// TwinCAT 3 PLC project Untitled1
// ProgramVersion: 3.1.4022.4
// libraries:
//   Tc2_MC2, * (Beckhoff Automation GmbH)
//   Tc2_Standard, * (Beckhoff Automation GmbH)
//   Tc2_System, * (Beckhoff Automation GmbH)
//   Tc3_Module, * (Beckhoff Automation GmbH)
// project tree:
//   GVLs/ GVL_IO.TcGVL
//   / PlcTask.TcTTO
//   POUs/ FB_Control.TcPOU, FB_Motion.TcPOU, MAIN.TcPOU
// real-time tasks:
//   TASK PlcTask: cycle T#10ms, priority 20, ADS port 350
// motion (NC):
//   TASK NC-Task 1 SAF: cycle T#2ms, priority 4, ADS port 501
//   TASK NC-Task 1 SVB: cycle T#10ms, priority 8, ADS port 511
//   AXIS Axis 1 (id 1)
//     Dynamic: Acceleration=12830.3, Deceleration=12830.3, Jerk=38490.9
//     Velo: RefSearch=85.5352783203125, RefSync=85.5352783203125, SlowManual=427.676391601563, FastManual=2566.05834960938, Fast=8553.52783203125, Maximum=8553.53
//     OtherSettings: AllowMotionCmdToSlave=true
//     encoder EncType=8
//       EncPara: ScaleFactorNumerator=100, ScaleFactorDenominator=1048576, MaxCount=#xffffffff
//     drive DrvType=9
//       DrvPara: MaxCount=#xffffffff, DriveControlDWord=#x00030100
//         Analog: VeloReferenz=9408.88061523438, VeloScale=1.02400649589962, ScaleFactorActTorque=0.1
//         TimeComp: TaskDelayCycles=1
//     controller CtrType=1
//       CtrPara: PriorControlFactor=1
//         Observer: BandWidth=20
//   AXIS Axis 2 (id 2)
//     Dynamic: Acceleration=12632.5, Deceleration=12632.5, Jerk=37897.6
//     Velo: RefSearch=84.2169026692708, RefSync=84.2169026692708, SlowManual=421.084513346354, FastManual=2526.50708007813, Fast=8421.69026692708, Maximum=8421.69
//     OtherSettings: AllowMotionCmdToSlave=true
//     encoder EncType=1
//       EncPara: ScaleFactorNumerator=100, ScaleFactorDenominator=1048576
//     drive DrvType=5
//       Analog: VeloReferenz=9263.85929361979, ScaleFactorActTorque=0.1
//       TimeComp: TaskDelayCycles=1
//     controller CtrType=1
//       CtrPara: PriorControlFactor=1
//         Observer: BandWidth=20
// I/O:
//   DEVICE Device 1 (EtherCAT), AmsNetId 169.254.89.106.2.1
//     Term 1 (EK1200) [EK1200-5000 EtherCAT Power supply (2A E-Bus)]
//       Term 2 (EL1004) [EL1004 4Ch. Dig. Input 24V, 3ms]
//       Term 3 (EL2004) [EL2004 4Ch. Dig. Output 24V, 0.5A]
//       Term 4 (EL3062) [EL3062 2Ch. Ana. Input 0-10V]
//       Term 5 (EL4002) [EL4002 2Ch. Ana. Output 0-10V, 12bit]
//       Term 6 (EK1110) [EK1110 EtherCAT extension]
//     Drive 7 (AX5203-0000-0210) [AX5203-0000-0210 EtherCAT Drive (SoE, 2 Ch.)]
// variable links:
//   NC-Task 1 SAF/Axes/Axis 1 <-> Device 1 (EtherCAT)/Drive 7 (AX5203-0000-0210)
//     Drive/Inputs/In/nDataIn1 <-> AT 1/Following distance
//     Drive/Inputs/In/nDcOutputTime <-> InfoData/DcOutputShift
//     Drive/Inputs/In/nState1 <-> AT 1/Drive status word @bit 8
//     Drive/Inputs/In/nState2 <-> AT 1/Drive status word
//     Drive/Inputs/In/nState4 @bit 1 <-> WcState/InputToggle
//     Drive/Inputs/In/nState4 <-> WcState/WcState
//     Drive/Outputs/Out/nCtrl1 <-> MDT 1/Master control word @bit 8
//     Drive/Outputs/Out/nDataOut1 <-> MDT 1/Position command value
//     Enc/Inputs/In/nDataIn1 <-> AT 1/Position feedback 1 value
//     Enc/Inputs/In/nDcInputTime <-> InfoData/DcInputShift
//     Enc/Inputs/In/nState4 @bit 1 <-> WcState/InputToggle
//     Enc/Inputs/In/nState4 <-> WcState/WcState
//   Untitled1/Untitled1 Instance <-> NC-Task 1 SAF/Axes/Axis 1
//     PlcTask Inputs/GVL_IO.Axis1.NcToPlc <-> Outputs/ToPlc
//     PlcTask Outputs/GVL_IO.Axis1.PlcToNc <-> Inputs/FromPlc

CONFIGURATION Untitled1
    RESOURCE PLC ON TwinCAT3
        TASK PlcTask(INTERVAL := T#10ms, PRIORITY := 20);
        PROGRAM MAIN WITH PlcTask : MAIN;
    END_RESOURCE
END_CONFIGURATION

// ---- GVLs/GVL_IO.TcGVL
VAR_GLOBAL
	

binput1 AT%I* :BOOL;

boutput1 AT%Q* :BOOL;

Axis1 :AXIS_REF;
Axis2 :AXIS_REF;

END_VAR

// ---- POUs/MAIN.TcPOU
PROGRAM MAIN
VAR
	FB_Control1: FB_Control;
	FB_Motion1: FB_Motion;

	button1: BOOL;
END_VAR





(*FB_Motion1(
	bStart:=binput1 , 
	bExecute:=main.FB_Control1.ProgEx , 
	bBusy=> , 
	bDone=> , 
	nPosition:=main.FB_Control1.position , 
	);
	*)
FB_Motion1(
	bMoveAbs	:=main.FB_Control1.ProgEx, 
	nPosition	:=main.FB_Control1.position , 
	bBusy		=> , 
	bDone		=> , 
	bStopEx		:=main.FB_Control1.StopState,
	bStopDone	=>  
	 );
	
FB_Control1(
	
button1:= button1  , 
ProcessDone:=, 
StopDone := main.FB_Motion1.bStopDone  , 
ProgEx=>
);

END_PROGRAM

// ---- POUs/FB_Control.TcPOU
FUNCTION_BLOCK FB_Control
VAR_INPUT
	button1: BOOL;
	ProcessDone: BOOL;
	StopDone: BOOL;
END_VAR
VAR_OUTPUT
	position: LREAL;
	ProgEx: BOOL;
	StopState: BOOL;
END_VAR
VAR
	nState: INT;
	TON1: TON;
	TON2: TON;
	TON3: TON;
	R_TRIG1: R_TRIG;
	F_TRIG1: F_TRIG;
END_VAR
VAR_IN_OUT
	
	
END_VAR



CASE nState OF
0:
	
	IF button1 THEN
		StopState:=FALSE;
		nState:=10;
	END_IF
10:
	nState:=15;
	position:=30000;
	progEx:=TRUE;

15:
	
IF ProcessDone THEN
	TON1(IN:=TRUE, PT:=T#1S , Q=> , ET=> );
	IF TON1.Q THEN
		nState:=19;
		TON1(IN:=FALSE);

	END_IF
END_IF

19:
	ProgEx:=FALSE;
	nState:=20;

20:
	position:=20000;
	nState	:=25;
	progEx	:=TRUE;


25:
IF ProcessDone THEN
		TON2(IN:=TRUE, PT:=T#4S , Q=> , ET=> );
	IF TON2.Q THEN
		nState:=26;
		TON2(IN:=FALSE);
	END_IF
END_IF

26:
	ProgEx:=FALSE;
	nState:=30;

30:
	position:=0;
	nState:=35;
	progEx:=TRUE;

35:
IF ProcessDone THEN
		TON3(IN:=TRUE, PT:=T#2S , Q=> , ET=> );
	IF TON3.Q THEN
		nState:=36;
		TON3(IN:=FALSE);
	END_IF
END_IF
36:
	
	ProgEx:=FALSE;
	nState:=0;

100:
	StopState:=TRUE;
	IF StopDone THEN
		nState:=0;
		TON1(IN:=FALSE);
		TON2(IN:=FALSE);
		TON3(IN:=FALSE);
		ProgEx:=FALSE;
		StopState:=FALSE;

END_IF
END_CASE
F_TRIG1(CLK:=button1 , Q=> );

IF F_TRIG1.Q THEN
	nState:=100;
END_IF

END_FUNCTION_BLOCK

// ---- POUs/FB_Motion.TcPOU
FUNCTION_BLOCK FB_Motion
VAR_INPUT
	bStart: BOOL;
	nPosition: LREAL;
	bStopEx: BOOL;
	bMoveAbs: BOOL;
END_VAR
VAR_OUTPUT
	bBusy: BOOL;
	bDone: BOOL;
	bStopDone: BOOL;
END_VAR
VAR
	MC_Power1: MC_Power;
	MC_MoveAbsolute1: MC_MoveAbsolute;
	MC_Stop1: MC_Stop;

END_VAR

MC_Power1(
	Axis:=Axis1 , 
	Enable:=TRUE , 
	Enable_Positive:=TRUE , 
	Enable_Negative:=TRUE , 
	Override:=100, 
	BufferMode:= , 
	Options:= , 
	Status=> , 
	Busy=> , 
	Active=> , 
	Error=> , 
	ErrorID=> );
	
	
	MC_MoveAbsolute1(
	Axis:= Axis1, 
	Execute:=bMoveAbs , 
	Position:=nPosition , 
	Velocity:= 8000, 
	Acceleration:= , 
	Deceleration:= , 
	Jerk:= , 
	BufferMode:= , 
	Options:= , 
	Done=>bDone , 
	Busy=>bBusy , 
	Active=> , 
	CommandAborted=> , 
	Error=> , 
	ErrorID=> );
	
			MC_Stop1(
	Axis:=Axis1 , 
	Execute:=bStopEx , 
	Deceleration:= , 
	Jerk:= , 
	Options:= , 
	Done=>bStopDone , 
	Busy=> , 
	Active=> , 
	CommandAborted=> , 
	Error=> , 
	ErrorID=> );

END_FUNCTION_BLOCK
